// TIA Portal project "FBM_Bordeau" (V17)

(* hardware
DEVICE "S7-1200 station_1"  S7-1200 Station
   slot 0: "Rack_0"  S7-1200 Rack  Rack  V1.0
   slot 1: "PLC_1"  CPU 1214C AC/DC/Rly  6ES7 214-1BG40-0XB0  V4.5
DEVICE "S7-1200 station_2"  S7-1200 Station
   slot 0: "Rack_0"  S7-1200 Rack  Rack  V1.0
   slot 1: "PLC_2"  CPU 1214C AC/DC/Rly  6ES7 214-1BG40-0XB0  V4.5
DEVICE "HMI_1"  KTP400 Basic PN
   slot 0: "HMI_1"  KTP400 Basic PN  6AV2 123-2DB03-0AX0  17.0.0.0
   slot 1: "HMI_RT_1"  KTP400 Basic PN  6AV2 123-2DB03-0AX0  17.0.0.0
   slot 5: "HMI_1.IE_CP_1"  PROFINET Interface  17.0.0.0
      slot 1: "PROFINET Interface_1"  PROFINET Interface
         slot 1: "Port_1"  Port
*)

// ===== PLC "PLC_1"  CPU 1214C AC/DC/Rly =====

VAR_GLOBAL   // PLC tag table "Default tag table"
   "VisiteurMax" AT %MW10 : Int;
   "Alerte1" AT %MW12 : Int;
   "Alerte2" AT %MW14 : Int;
   "Occupation" AT %MW16 : Int;
   "BitAlerte1" AT %M50.0 : Bool;
   "BitAlerte2" AT %M50.1 : Bool;
   "BitNoAlerte" AT %M50.2 : Bool;
   "AnimationCarre" AT %MW18 : Int;
   "BitModifier" AT %M50.3 : Bool;
   "BitEnregistrer" AT %M50.4 : Bool;
   "BitAnnuler" AT %M50.5 : Bool;
   "AutoriseModifier" AT %M50.6 : Bool;
   "AutoriseEnregistrer" AT %M50.7 : Bool;
   "AutoriseAnnuler" AT %M51.0 : Bool;
   "FM_1" AT %M60.0 : Bool;
   "FM_2" AT %M60.1 : Bool;
   "Up" AT %M60.2 : Bool;
   "Down" AT %M60.3 : Bool;
   "FM_3" AT %M60.4 : Bool;
   "FM_4" AT %M60.5 : Bool;
   "RealOccupation" AT %MD100 : Real;
   "RealAlerte1" AT %MD104 : Real;
   "RealAlerte2" AT %MD108 : Real;
   "RealVisiteurMax" AT %MD112 : Real;
   "Tag_5" AT %MD116 : Real;
   "Tag_6" AT %MD120 : DWord;
   "FM_7" AT %M60.6 : Bool;
   "Tag_8" AT %MD122 : Real;
   "FM_9" AT %M60.7 : Bool;
   "OldVisiteurMax" AT %MW20 : Int;
   "PourcentageMax" AT %MD126 : Real;
   "PourcentageMin" AT %MD130 : Real;
   "IR1_COULOIR_1" AT %I0.0 : Bool;
   "COMPTEUR_E_COULOIR_1" AT %I0.1 : Bool;
   "COMPTEUR_S_COULOIR_1" AT %I0.2 : Bool;
   "IR1_COULOIR_2" AT %I0.3 : Bool;
   "COMPTEUR_E_COULOIR_2" AT %I0.4 : Bool;
   "COMPTEUR_S_COULOIR_2" AT %I0.5 : Bool;
   "IR1_COULOIR_3" AT %I0.6 : Bool;
   "COMPTEUR_E_COULOIR_3" AT %I0.7 : Bool;
   "COMPTEUR_S_COULOIR_3" AT %I1.0 : Bool;
   "IR1_COULOIR_4" AT %I1.1 : Bool;
   "COMPTEUR_E_COULOIR_4" AT %I1.2 : Bool;
   "COMPTEUR_S_COULOIR_4" AT %I1.3 : Bool;
   "RESERVE1" AT %I1.4 : Bool;
   "RESERVE2" AT %I1.5 : Bool;
   "COMMANDE_O_COULOIR_1" AT %Q0.0 : Bool;
   "COMMANDE_O_COULOIR_2" AT %Q0.1 : Bool;
   "COMMANDE_O_COULOIR_3" AT %Q0.2 : Bool;
   "COMMANDE_O_COULOIR_4" AT %Q0.3 : Bool;
   "COMMANDE_O_COULOIR_5" AT %Q0.4 : Bool;
   "COMMANDE_O_COULOIR_6" AT %Q0.5 : Bool;
   "COMMANDE_O_COULOIR_7" AT %Q0.6 : Bool;
   "RESERVE_SORTIE_8" AT %Q0.7 : Bool;
   "Sortie8" AT %Q1.0 : Bool;
   "Sortie9" AT %Q1.1 : Bool;
   "Clock_Byte" AT %MB0 : Byte;
   "Clock_10Hz" AT %M0.0 : Bool;
   "Clock_5Hz" AT %M0.1 : Bool;
   "Clock_2.5Hz" AT %M0.2 : Bool;
   "Clock_2Hz" AT %M0.3 : Bool;
   "Clock_1.25Hz" AT %M0.4 : Bool;
   "Clock_1Hz" AT %M0.5 : Bool;
   "Clock_0.625Hz" AT %M0.6 : Bool;
   "Clock_0.5Hz" AT %M0.7 : Bool;
   "PLC1_ImageEntree1" AT %M70.0 : Bool;
   "PLC1_ImageEntree2" AT %M70.1 : Bool;
   "PLC1_ImageEntree3" AT %M70.2 : Bool;
   "PLC1_ImageEntree4" AT %M70.3 : Bool;
   "PLC1_ImageEntree5" AT %M70.4 : Bool;
   "PLC1_ImageEntree6" AT %M70.5 : Bool;
   "PLC1_ImageEntree7" AT %M70.6 : Bool;
   "PLC1_ImageEntree8" AT %M70.7 : Bool;
   "PLC1_ImageEntree9" AT %M71.0 : Bool;
   "PLC1_ImageEntree10" AT %M71.1 : Bool;
   "PLC1_ImageEntree11" AT %M71.2 : Bool;
   "PLC1_ImageEntree12" AT %M71.3 : Bool;
   "PLC1_ImageEntree13" AT %M71.4 : Bool;
   "PLC1_ImageEntree0" AT %M71.5 : Bool;
   "SynthesEntree" AT %M71.6 : Bool;
   "SyntheseSortie" AT %M71.7 : Bool;
   "FM_SyntheseEntree" AT %M72.0 : Bool;
   "FM_SyntheseSortie" AT %M72.1 : Bool;
   "FM_IR1_C5" AT %M72.2 : Bool;
   "FM_IR1_C6" AT %M72.3 : Bool;
   "FM_IR1_C7" AT %M72.4 : Bool;
   "FM_IR1_C1" AT %M73.2 : Bool;
   "FM_IR1_C2" AT %M73.3 : Bool;
   "FM_IR1_C3" AT %M73.4 : Bool;
   "FM_IR1_C4" AT %M73.5 : Bool;
   "Tag_1" AT %M80.0 : Bool;
   "PLC1_ImageSortie0" AT %M73.6 : Bool;
   "PLC1_ImageSortie1" AT %M73.7 : Bool;
   "PLC1_ImageSortie2" AT %M74.0 : Bool;
   "PLC1_ImageSortie3" AT %M74.1 : Bool;
   "PLC1_ImageSortie4" AT %M74.2 : Bool;
   "PLC1_ImageSortie5" AT %M74.3 : Bool;
   "PLC1_ImageSortie6" AT %M74.4 : Bool;
   "PLC2_ImageSortie0" AT %M74.5 : Bool;
   "PLC2_ImageSortie1" AT %M74.6 : Bool;
   "PLC2_ImageSortie2" AT %M74.7 : Bool;
   "PLC2_ImageSortie3" AT %M75.0 : Bool;
   "PLC2_ImageSortie4" AT %M75.1 : Bool;
   "PLC2_ImageSortie5" AT %M75.2 : Bool;
   "PLC2_ImageSortie6" AT %M75.3 : Bool;
   "Tag_2" AT %M100.0 : Bool;
   "Tag_3" AT %M100.1 : Bool;
   "Tag_4" AT %M100.2 : Bool;
   "Tag_7" AT %M100.3 : Bool;
   "TEST_SORTIE" AT %M100.4 : Bool;
   "TEST_ENTREE" AT %M100.5 : Bool;
   "ResetOccupation" AT %M100.6 : Bool;
   "Tag_9" AT %M100.7 : Bool;
   "FM_COUNT_S1" AT %M103.1 : Bool;
   "Memore_Cmpt_SortieC1" AT %M101.1 : Bool;
   "TempoIR1" AT %M102.1 : Bool;
   "Tag_11" AT %I1.6 : Bool;
   "Memore_Cmpt_SortieC2" AT %M101.2 : Bool;
   "Memore_Cmpt_SortieC3" AT %M101.3 : Bool;
   "Memore_Cmpt_SortieC4" AT %M101.4 : Bool;
   "Memore_Cmpt_SortieC5" AT %M101.5 : Bool;
   "Memore_Cmpt_SortieC6" AT %M101.6 : Bool;
   "Memore_Cmpt_SortieC7" AT %M101.7 : Bool;
   "TempoIR2" AT %M102.2 : Bool;
   "TempoIR3" AT %M102.3 : Bool;
   "TempoIR4" AT %M102.4 : Bool;
   "TempoIR5" AT %M102.5 : Bool;
   "TempoIR6" AT %M102.6 : Bool;
   "TempoIR7" AT %M102.7 : Bool;
   "FM_COUNT_S2" AT %M103.2 : Bool;
   "FM_COUNT_S3" AT %M103.3 : Bool;
   "FM_COUNT_S4" AT %M103.4 : Bool;
   "FM_COUNT_S5" AT %M103.5 : Bool;
   "FM_COUNT_S6" AT %M103.6 : Bool;
   "FM_COUNT_S7" AT %M103.7 : Bool;
END_VAR

DATA_BLOCK "PLC1_DB_Bool"   // DB1
{ S7_Optimized_Access := 'FALSE' }
VERSION : 0.1
   VAR
      FM_2 : Bool;
      Up : Bool;
      FM_4 : Bool;
      FM_1 : Bool;
      AutoriseAnnuler : Bool;
      AutoriseEnregistrer : Bool;
      AutoriseModifier : Bool;
      BitAnnuler : Bool;
      Down : Bool;
      BitEnregistrer : Bool;
      BitNoAlerte : Bool;
      BitAlerte2 : Bool;
      BitAlerte1 : Bool;
      FM_7 : Bool;
      FM_9 : Bool;
      BitModifier : Bool;
      FM_3 : Bool;
   END_VAR
BEGIN
END_DATA_BLOCK

DATA_BLOCK "PLC1_DB_Real"   // DB2
{ S7_Optimized_Access := 'FALSE' }
VERSION : 0.1
   VAR
      RealOccupation : Real;
      RealAlerte1 : Real;
      RealAlerte2 : Real;
      RealVisiteurMax : Real;
      Tag_5 : Real;
      Tag_8 : Real;
      PourcentageMax : Real;
      PourcentageMin : Real;
   END_VAR
BEGIN
END_DATA_BLOCK

DATA_BLOCK "PLC1_DB_Int"   // DB3
{ S7_Optimized_Access := 'FALSE' }
VERSION : 0.1
   VAR
      OldVisiteurMax : Int;
      VisiteurMax : Int;
      AnimationCarre : Int;
      Occupation : Int;
      Alerte2 : Int;
      Alerte1 : Int;
   END_VAR
BEGIN
END_DATA_BLOCK

DATA_BLOCK "PLC1_DB_TO_GET"   // DB4
{ S7_Optimized_Access := 'FALSE' }
VERSION : 0.1
   VAR
      IR1_COULOIR_5 : Bool;
      COMPTEUR_E_COULOIR_5 : Bool;
      COMPTEUR_S_COULOIR_5 : Bool;
      IR1_COULOIR_6 : Bool;
      COMPTEUR_E_COULOIR_6 : Bool;
      COMPTEUR_S_COULOIR_6 : Bool;
      IR1_COULOIR_7 : Bool;
      COMPTEUR_E_COULOIR_7 : Bool;
      COMPTEUR_S_COULOIR_7 : Bool;
      RESERVE_ENTREE_1 : Bool;
      RESERVE_ENTREE_2 : Bool;
      RESERVE_ENTREE_3 : Bool;
      RESERVE_ENTREE_4 : Bool;
      RESERVE_ENTREE_5 : Bool;
      RESERVE_SORTIE_0 : Bool;
      RESERVE_SORTIE_1 : Bool;
      RESERVE_SORTIE_2 : Bool;
      RESERVE_SORTIE_3 : Bool;
      RESERVE_SORTIE_4 : Bool;
      RESERVE_SORTIE_5 : Bool;
      RESERVE_SORTIE_6 : Bool;
   END_VAR
BEGIN
END_DATA_BLOCK

DATA_BLOCK "PLC1_DB_TO_PUT"   // DB6
{ S7_Optimized_Access := 'FALSE' }
VERSION : 0.1
   VAR
      Entree0 : Bool;
      Entree1 : Bool;
      Entree2 : Bool;
      Entree3 : Bool;
      Entree4 : Bool;
      Entree5 : Bool;
      Entree6 : Bool;
      Entree7 : Bool;
      Entree8 : Bool;
      Entree9 : Bool;
      Entree10 : Bool;
      Entree11 : Bool;
      Entree12 : Bool;
      Entree13 : Bool;
      Sortie0 : Bool;
      Sortie1 : Bool;
      Sortie2 : Bool;
      Sortie3 : Bool;
      Sortie4 : Bool;
      Sortie5 : Bool;
      Sortie6 : Bool;
   END_VAR
BEGIN
END_DATA_BLOCK

// folder: System blocks/Program resources

DATA_BLOCK "IEC_Timer_0_DB"   // DB8
{ S7_Optimized_Access := 'TRUE' }
AUTHOR : Simatic
FAMILY : IEC
NAME : IEC_TMR
VERSION : 1.0
// stored: InstanceOfName IEC_TIMER
"IEC_TIMER"
BEGIN
END_DATA_BLOCK

DATA_BLOCK "IEC_Timer_0_DB_2"   // DB9
{ S7_Optimized_Access := 'TRUE' }
AUTHOR : Simatic
FAMILY : IEC
NAME : IEC_TMR
VERSION : 1.0
// stored: InstanceOfName IEC_TIMER
"IEC_TIMER"
BEGIN
END_DATA_BLOCK

DATA_BLOCK "IEC_Timer_0_DB_3"   // DB10
{ S7_Optimized_Access := 'TRUE' }
AUTHOR : Simatic
FAMILY : IEC
NAME : IEC_TMR
VERSION : 1.0
// stored: InstanceOfName IEC_TIMER
"IEC_TIMER"
BEGIN
END_DATA_BLOCK

DATA_BLOCK "IEC_Timer_0_DB_4"   // DB11
{ S7_Optimized_Access := 'TRUE' }
AUTHOR : Simatic
FAMILY : IEC
NAME : IEC_TMR
VERSION : 1.0
// stored: InstanceOfName IEC_TIMER
"IEC_TIMER"
BEGIN
END_DATA_BLOCK

DATA_BLOCK "IEC_Timer_0_DB_5"   // DB12
{ S7_Optimized_Access := 'TRUE' }
AUTHOR : Simatic
FAMILY : IEC
NAME : IEC_TMR
VERSION : 1.0
// stored: InstanceOfName IEC_TIMER
"IEC_TIMER"
BEGIN
END_DATA_BLOCK

DATA_BLOCK "IEC_Timer_0_DB_6"   // DB13
{ S7_Optimized_Access := 'TRUE' }
AUTHOR : Simatic
FAMILY : IEC
NAME : IEC_TMR
VERSION : 1.0
// stored: InstanceOfName IEC_TIMER
"IEC_TIMER"
BEGIN
END_DATA_BLOCK

DATA_BLOCK "IEC_Timer_0_DB_7"   // DB14
{ S7_Optimized_Access := 'TRUE' }
AUTHOR : Simatic
FAMILY : IEC
NAME : IEC_TMR
VERSION : 1.0
// stored: InstanceOfName IEC_TIMER
"IEC_TIMER"
BEGIN
END_DATA_BLOCK

DATA_BLOCK "IEC_Timer_0_DB_8"   // DB15
{ S7_Optimized_Access := 'TRUE' }
AUTHOR : Simatic
FAMILY : IEC
NAME : IEC_TMR
VERSION : 1.0
// stored: InstanceOfName IEC_TIMER
"IEC_TIMER"
BEGIN
END_DATA_BLOCK

DATA_BLOCK "IEC_Timer_0_DB_1"   // DB16
{ S7_Optimized_Access := 'TRUE' }
AUTHOR : Simatic
FAMILY : IEC
NAME : IEC_TMR
VERSION : 1.0
// stored: InstanceOfName IEC_TIMER
"IEC_TIMER"
BEGIN
END_DATA_BLOCK

DATA_BLOCK "IEC_Timer_0_DB_9"   // DB17
{ S7_Optimized_Access := 'TRUE' }
AUTHOR : Simatic
FAMILY : IEC
NAME : IEC_TMR
VERSION : 1.0
// stored: InstanceOfName IEC_TIMER
"IEC_TIMER"
BEGIN
END_DATA_BLOCK

DATA_BLOCK "IEC_Timer_0_DB_10"   // DB18
{ S7_Optimized_Access := 'TRUE' }
AUTHOR : Simatic
FAMILY : IEC
NAME : IEC_TMR
VERSION : 1.0
// stored: InstanceOfName IEC_TIMER
"IEC_TIMER"
BEGIN
END_DATA_BLOCK

DATA_BLOCK "IEC_Timer_0_DB_11"   // DB19
{ S7_Optimized_Access := 'TRUE' }
AUTHOR : Simatic
FAMILY : IEC
NAME : IEC_TMR
VERSION : 1.0
// stored: InstanceOfName IEC_TIMER
"IEC_TIMER"
BEGIN
END_DATA_BLOCK

DATA_BLOCK "IEC_Timer_0_DB_12"   // DB20
{ S7_Optimized_Access := 'TRUE' }
AUTHOR : Simatic
FAMILY : IEC
NAME : IEC_TMR
VERSION : 1.0
// stored: InstanceOfName IEC_TIMER
"IEC_TIMER"
BEGIN
END_DATA_BLOCK

DATA_BLOCK "IEC_Timer_0_DB_13"   // DB21
{ S7_Optimized_Access := 'TRUE' }
AUTHOR : Simatic
FAMILY : IEC
NAME : IEC_TMR
VERSION : 1.0
// stored: InstanceOfName IEC_TIMER
"IEC_TIMER"
BEGIN
END_DATA_BLOCK

DATA_BLOCK "IEC_Timer_0_DB_14"   // DB22
{ S7_Optimized_Access := 'TRUE' }
AUTHOR : Simatic
FAMILY : IEC
NAME : IEC_TMR
VERSION : 1.0
// stored: InstanceOfName IEC_TIMER
"IEC_TIMER"
BEGIN
END_DATA_BLOCK

DATA_BLOCK "IEC_Timer_0_DB_15"   // DB23
{ S7_Optimized_Access := 'TRUE' }
AUTHOR : Simatic
FAMILY : IEC
NAME : IEC_TMR
VERSION : 1.0
// stored: InstanceOfName IEC_TIMER
"IEC_TIMER"
BEGIN
END_DATA_BLOCK

DATA_BLOCK "IEC_Timer_0_DB_16"   // DB24
{ S7_Optimized_Access := 'TRUE' }
AUTHOR : Simatic
FAMILY : IEC
NAME : IEC_TMR
VERSION : 1.0
// stored: InstanceOfName IEC_TIMER
"IEC_TIMER"
BEGIN
END_DATA_BLOCK

DATA_BLOCK "IEC_Timer_0_DB_17"   // DB25
{ S7_Optimized_Access := 'TRUE' }
AUTHOR : Simatic
FAMILY : IEC
NAME : IEC_TMR
VERSION : 1.0
// stored: InstanceOfName IEC_TIMER
"IEC_TIMER"
BEGIN
END_DATA_BLOCK

DATA_BLOCK "IEC_Timer_0_DB_18"   // DB26
{ S7_Optimized_Access := 'TRUE' }
AUTHOR : Simatic
FAMILY : IEC
NAME : IEC_TMR
VERSION : 1.0
// stored: InstanceOfName IEC_TIMER
"IEC_TIMER"
BEGIN
END_DATA_BLOCK

DATA_BLOCK "IEC_Timer_0_DB_19"   // DB27
{ S7_Optimized_Access := 'TRUE' }
AUTHOR : Simatic
FAMILY : IEC
NAME : IEC_TMR
VERSION : 1.0
// stored: InstanceOfName IEC_TIMER
"IEC_TIMER"
BEGIN
END_DATA_BLOCK

// folder: (top level)

FUNCTION "PLC1_Get_Put_Value_PLC2" : Void   // FC1, LAD
{ S7_Optimized_Access := 'TRUE' }
VERSION : 0.1
BEGIN

REGION Network 1
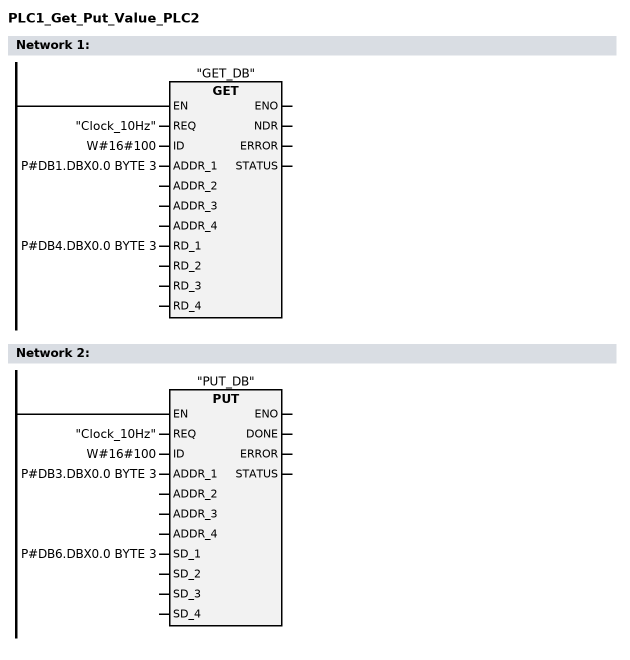
   "GET_DB"(REQ := "Clock_10Hz", ID := W#16#100, ADDR_1 := P#DB1.DBX0.0 BYTE 3, RD_1 := P#DB4.DBX0.0 BYTE 3);   // GET
END_REGION

REGION Network 2
   "PUT_DB"(REQ := "Clock_10Hz", ID := W#16#100, ADDR_1 := P#DB3.DBX0.0 BYTE 3, SD_1 := P#DB6.DBX0.0 BYTE 3);   // PUT
END_REGION
END_FUNCTION

FUNCTION "PLC1_ImageEntree" : Void   // FC2, LAD
{ S7_Optimized_Access := 'TRUE' }
VERSION : 0.1
BEGIN

REGION Network 1: SYNTHESE ENTREE SUR SITE
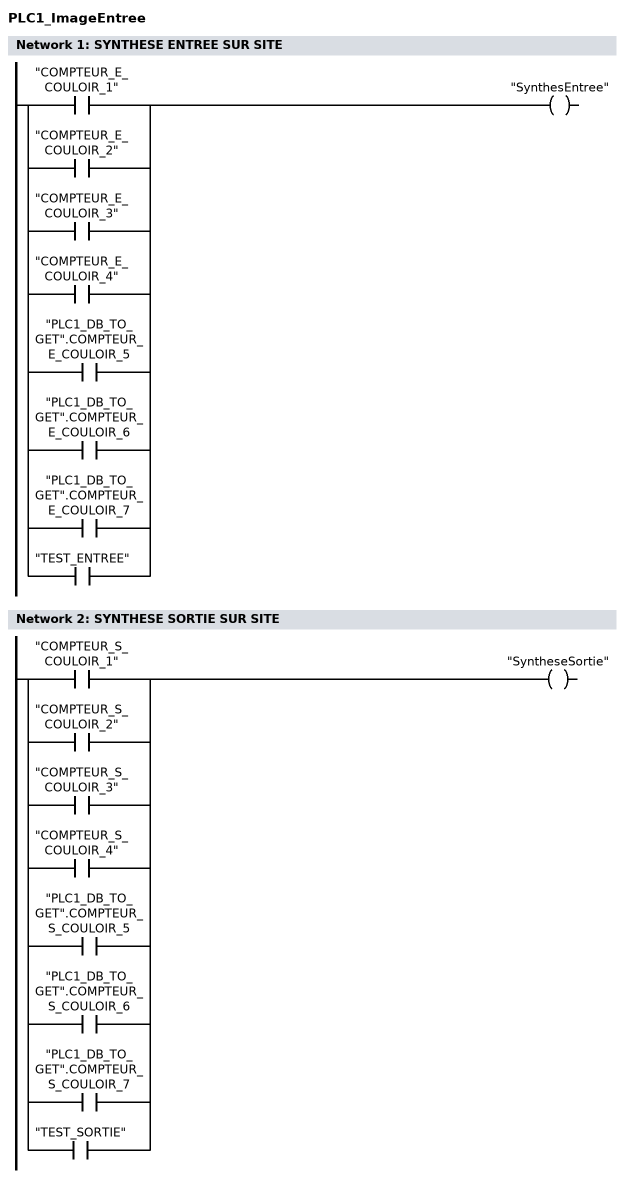
   RUNG wire#powerrail
      Contact( "COMPTEUR_E_COULOIR_1" )
      wire#w1
      Coil( "SynthesEntree" )
   END_RUNG
   RUNG wire#powerrail
      Contact( "COMPTEUR_E_COULOIR_2" )
   END_RUNG wire#w1
   RUNG wire#powerrail
      Contact( "COMPTEUR_E_COULOIR_3" )
   END_RUNG wire#w1
   RUNG wire#powerrail
      Contact( "COMPTEUR_E_COULOIR_4" )
   END_RUNG wire#w1
   RUNG wire#powerrail
      Contact( "PLC1_DB_TO_GET".COMPTEUR_E_COULOIR_5 )
   END_RUNG wire#w1
   RUNG wire#powerrail
      Contact( "PLC1_DB_TO_GET".COMPTEUR_E_COULOIR_6 )
   END_RUNG wire#w1
   RUNG wire#powerrail
      Contact( "PLC1_DB_TO_GET".COMPTEUR_E_COULOIR_7 )
   END_RUNG wire#w1
   RUNG wire#powerrail
      Contact( "TEST_ENTREE" )
   END_RUNG wire#w1
   // the same network as SCL:
   "SynthesEntree" := "COMPTEUR_E_COULOIR_1" OR "COMPTEUR_E_COULOIR_2" OR "COMPTEUR_E_COULOIR_3" OR "COMPTEUR_E_COULOIR_4" OR "PLC1_DB_TO_GET".COMPTEUR_E_COULOIR_5 OR "PLC1_DB_TO_GET".COMPTEUR_E_COULOIR_6 OR "PLC1_DB_TO_GET".COMPTEUR_E_COULOIR_7 OR "TEST_ENTREE";
END_REGION

REGION Network 2: SYNTHESE SORTIE SUR SITE
   RUNG wire#powerrail
      Contact( "COMPTEUR_S_COULOIR_1" )
      wire#w1
      Coil( "SyntheseSortie" )
   END_RUNG
   RUNG wire#powerrail
      Contact( "COMPTEUR_S_COULOIR_2" )
   END_RUNG wire#w1
   RUNG wire#powerrail
      Contact( "COMPTEUR_S_COULOIR_3" )
   END_RUNG wire#w1
   RUNG wire#powerrail
      Contact( "COMPTEUR_S_COULOIR_4" )
   END_RUNG wire#w1
   RUNG wire#powerrail
      Contact( "PLC1_DB_TO_GET".COMPTEUR_S_COULOIR_5 )
   END_RUNG wire#w1
   RUNG wire#powerrail
      Contact( "PLC1_DB_TO_GET".COMPTEUR_S_COULOIR_6 )
   END_RUNG wire#w1
   RUNG wire#powerrail
      Contact( "PLC1_DB_TO_GET".COMPTEUR_S_COULOIR_7 )
   END_RUNG wire#w1
   RUNG wire#powerrail
      Contact( "TEST_SORTIE" )
   END_RUNG wire#w1
   // the same network as SCL:
   "SyntheseSortie" := "COMPTEUR_S_COULOIR_1" OR "COMPTEUR_S_COULOIR_2" OR "COMPTEUR_S_COULOIR_3" OR "COMPTEUR_S_COULOIR_4" OR "PLC1_DB_TO_GET".COMPTEUR_S_COULOIR_5 OR "PLC1_DB_TO_GET".COMPTEUR_S_COULOIR_6 OR "PLC1_DB_TO_GET".COMPTEUR_S_COULOIR_7 OR "TEST_SORTIE";
END_REGION
END_FUNCTION

ORGANIZATION_BLOCK "PLC1_Main"   // OB1, LAD, ProgramCycle
TITLE = "Main Program Sweep (Cycle)"
{ S7_Optimized_Access := 'TRUE' }
VERSION : 0.1
   VAR_INPUT
      Initial_Call : Bool;   // Initial call of this OB
      Remanence : Bool;   // =True, if remanent data are available
   END_VAR
   VAR_TEMP   // added for the SCL form of the ladder/FBD networks
      _w1 : Bool;
      _w2 : Bool;
      _w3 : Bool;
      _w4 : Bool;
   END_VAR
BEGIN

REGION Network 1
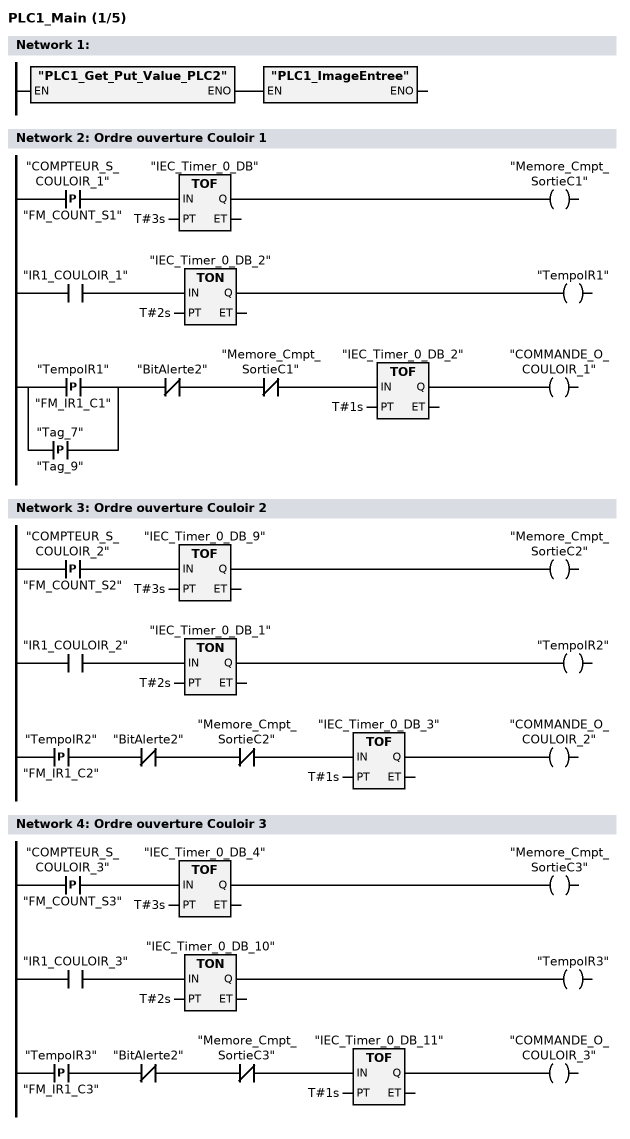
   RUNG wire#powerrail
      "PLC1_Get_Put_Value_PLC2"()
      "PLC1_ImageEntree"()
   END_RUNG
   // the same network as SCL:
   "PLC1_Get_Put_Value_PLC2"(ENO => #_w1);
   IF #_w1 THEN "PLC1_ImageEntree"(); END_IF;
END_REGION

REGION Network 2: Ordre ouverture Couloir 1
   #_w1 := "COMPTEUR_S_COULOIR_1" AND NOT "FM_COUNT_S1";   // rising edge of "COMPTEUR_S_COULOIR_1"
   "FM_COUNT_S1" := "COMPTEUR_S_COULOIR_1";
   "IEC_Timer_0_DB".TOF(IN := #_w1, PT := T#3s);
   "Memore_Cmpt_SortieC1" := "IEC_Timer_0_DB".Q;
   "IEC_Timer_0_DB_2".TON(IN := "IR1_COULOIR_1", PT := T#2s);
   "TempoIR1" := "IEC_Timer_0_DB_2".Q;
   #_w2 := "TempoIR1" AND NOT "FM_IR1_C1";   // rising edge of "TempoIR1"
   "FM_IR1_C1" := "TempoIR1";
   #_w3 := "Tag_7" AND NOT "Tag_9";   // rising edge of "Tag_7"
   "Tag_9" := "Tag_7";
   "IEC_Timer_0_DB_2".TOF(IN := (#_w2 OR #_w3) AND NOT "BitAlerte2" AND NOT "Memore_Cmpt_SortieC1", PT := T#1s);
   "COMMANDE_O_COULOIR_1" := "IEC_Timer_0_DB_2".Q;
END_REGION

REGION Network 3: Ordre ouverture Couloir 2
   #_w1 := "COMPTEUR_S_COULOIR_2" AND NOT "FM_COUNT_S2";   // rising edge of "COMPTEUR_S_COULOIR_2"
   "FM_COUNT_S2" := "COMPTEUR_S_COULOIR_2";
   "IEC_Timer_0_DB_9".TOF(IN := #_w1, PT := T#3s);
   "Memore_Cmpt_SortieC2" := "IEC_Timer_0_DB_9".Q;
   "IEC_Timer_0_DB_1".TON(IN := "IR1_COULOIR_2", PT := T#2s);
   "TempoIR2" := "IEC_Timer_0_DB_1".Q;
   #_w2 := "TempoIR2" AND NOT "FM_IR1_C2";   // rising edge of "TempoIR2"
   "FM_IR1_C2" := "TempoIR2";
   "IEC_Timer_0_DB_3".TOF(IN := #_w2 AND NOT "BitAlerte2" AND NOT "Memore_Cmpt_SortieC2", PT := T#1s);
   "COMMANDE_O_COULOIR_2" := "IEC_Timer_0_DB_3".Q;
END_REGION

REGION Network 4: Ordre ouverture Couloir 3
   #_w1 := "COMPTEUR_S_COULOIR_3" AND NOT "FM_COUNT_S3";   // rising edge of "COMPTEUR_S_COULOIR_3"
   "FM_COUNT_S3" := "COMPTEUR_S_COULOIR_3";
   "IEC_Timer_0_DB_4".TOF(IN := #_w1, PT := T#3s);
   "Memore_Cmpt_SortieC3" := "IEC_Timer_0_DB_4".Q;
   "IEC_Timer_0_DB_10".TON(IN := "IR1_COULOIR_3", PT := T#2s);
   "TempoIR3" := "IEC_Timer_0_DB_10".Q;
   #_w2 := "TempoIR3" AND NOT "FM_IR1_C3";   // rising edge of "TempoIR3"
   "FM_IR1_C3" := "TempoIR3";
   "IEC_Timer_0_DB_11".TOF(IN := #_w2 AND NOT "BitAlerte2" AND NOT "Memore_Cmpt_SortieC3", PT := T#1s);
   "COMMANDE_O_COULOIR_3" := "IEC_Timer_0_DB_11".Q;
END_REGION

REGION Network 5: Ordre ouverture Couloir 4
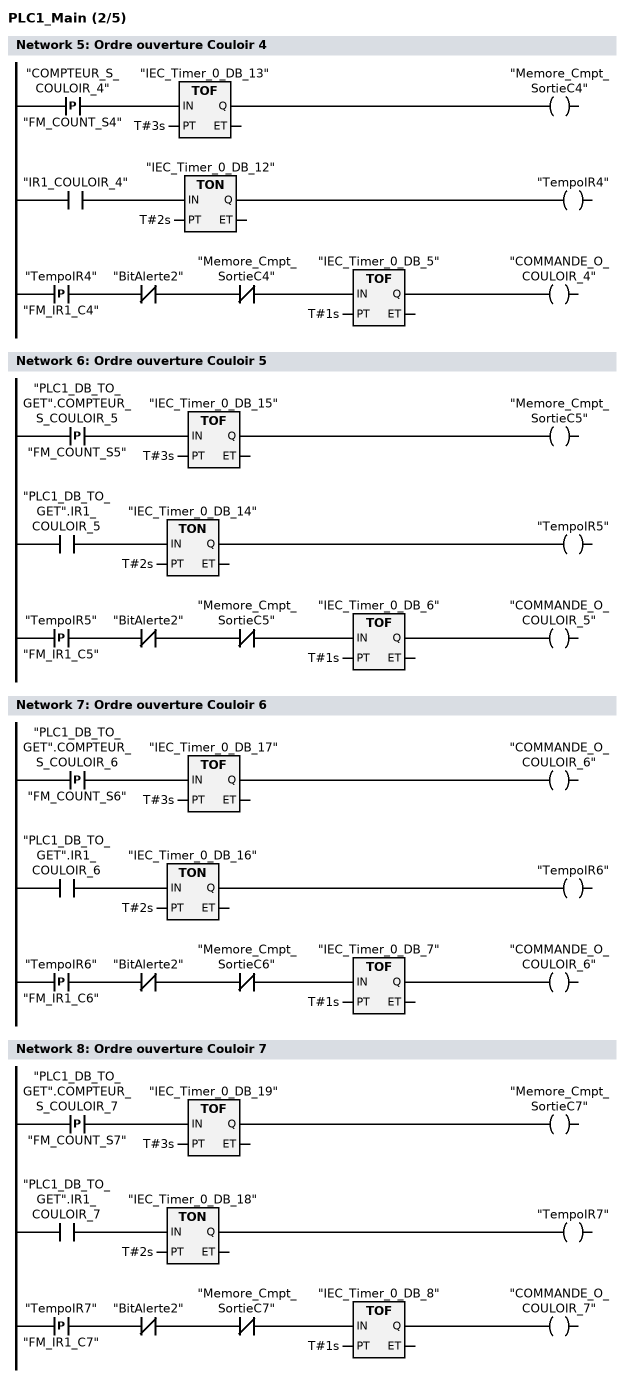
   #_w1 := "COMPTEUR_S_COULOIR_4" AND NOT "FM_COUNT_S4";   // rising edge of "COMPTEUR_S_COULOIR_4"
   "FM_COUNT_S4" := "COMPTEUR_S_COULOIR_4";
   "IEC_Timer_0_DB_13".TOF(IN := #_w1, PT := T#3s);
   "Memore_Cmpt_SortieC4" := "IEC_Timer_0_DB_13".Q;
   "IEC_Timer_0_DB_12".TON(IN := "IR1_COULOIR_4", PT := T#2s);
   "TempoIR4" := "IEC_Timer_0_DB_12".Q;
   #_w2 := "TempoIR4" AND NOT "FM_IR1_C4";   // rising edge of "TempoIR4"
   "FM_IR1_C4" := "TempoIR4";
   "IEC_Timer_0_DB_5".TOF(IN := #_w2 AND NOT "BitAlerte2" AND NOT "Memore_Cmpt_SortieC4", PT := T#1s);
   "COMMANDE_O_COULOIR_4" := "IEC_Timer_0_DB_5".Q;
END_REGION

REGION Network 6: Ordre ouverture Couloir 5
   #_w1 := "PLC1_DB_TO_GET".COMPTEUR_S_COULOIR_5 AND NOT "FM_COUNT_S5";   // rising edge of "PLC1_DB_TO_GET".COMPTEUR_S_COULOIR_5
   "FM_COUNT_S5" := "PLC1_DB_TO_GET".COMPTEUR_S_COULOIR_5;
   "IEC_Timer_0_DB_15".TOF(IN := #_w1, PT := T#3s);
   "Memore_Cmpt_SortieC5" := "IEC_Timer_0_DB_15".Q;
   "IEC_Timer_0_DB_14".TON(IN := "PLC1_DB_TO_GET".IR1_COULOIR_5, PT := T#2s);
   "TempoIR5" := "IEC_Timer_0_DB_14".Q;
   #_w2 := "TempoIR5" AND NOT "FM_IR1_C5";   // rising edge of "TempoIR5"
   "FM_IR1_C5" := "TempoIR5";
   "IEC_Timer_0_DB_6".TOF(IN := #_w2 AND NOT "BitAlerte2" AND NOT "Memore_Cmpt_SortieC5", PT := T#1s);
   "COMMANDE_O_COULOIR_5" := "IEC_Timer_0_DB_6".Q;
END_REGION

REGION Network 7: Ordre ouverture Couloir 6
   #_w1 := "PLC1_DB_TO_GET".COMPTEUR_S_COULOIR_6 AND NOT "FM_COUNT_S6";   // rising edge of "PLC1_DB_TO_GET".COMPTEUR_S_COULOIR_6
   "FM_COUNT_S6" := "PLC1_DB_TO_GET".COMPTEUR_S_COULOIR_6;
   "IEC_Timer_0_DB_17".TOF(IN := #_w1, PT := T#3s);
   "COMMANDE_O_COULOIR_6" := "IEC_Timer_0_DB_17".Q;
   "IEC_Timer_0_DB_16".TON(IN := "PLC1_DB_TO_GET".IR1_COULOIR_6, PT := T#2s);
   "TempoIR6" := "IEC_Timer_0_DB_16".Q;
   #_w2 := "TempoIR6" AND NOT "FM_IR1_C6";   // rising edge of "TempoIR6"
   "FM_IR1_C6" := "TempoIR6";
   "IEC_Timer_0_DB_7".TOF(IN := #_w2 AND NOT "BitAlerte2" AND NOT "Memore_Cmpt_SortieC6", PT := T#1s);
   "COMMANDE_O_COULOIR_6" := "IEC_Timer_0_DB_7".Q;
END_REGION

REGION Network 8: Ordre ouverture Couloir 7
   #_w1 := "PLC1_DB_TO_GET".COMPTEUR_S_COULOIR_7 AND NOT "FM_COUNT_S7";   // rising edge of "PLC1_DB_TO_GET".COMPTEUR_S_COULOIR_7
   "FM_COUNT_S7" := "PLC1_DB_TO_GET".COMPTEUR_S_COULOIR_7;
   "IEC_Timer_0_DB_19".TOF(IN := #_w1, PT := T#3s);
   "Memore_Cmpt_SortieC7" := "IEC_Timer_0_DB_19".Q;
   "IEC_Timer_0_DB_18".TON(IN := "PLC1_DB_TO_GET".IR1_COULOIR_7, PT := T#2s);
   "TempoIR7" := "IEC_Timer_0_DB_18".Q;
   #_w2 := "TempoIR7" AND NOT "FM_IR1_C7";   // rising edge of "TempoIR7"
   "FM_IR1_C7" := "TempoIR7";
   "IEC_Timer_0_DB_8".TOF(IN := #_w2 AND NOT "BitAlerte2" AND NOT "Memore_Cmpt_SortieC7", PT := T#1s);
   "COMMANDE_O_COULOIR_7" := "IEC_Timer_0_DB_8".Q;
END_REGION

REGION Network 9: Active Alerte 1
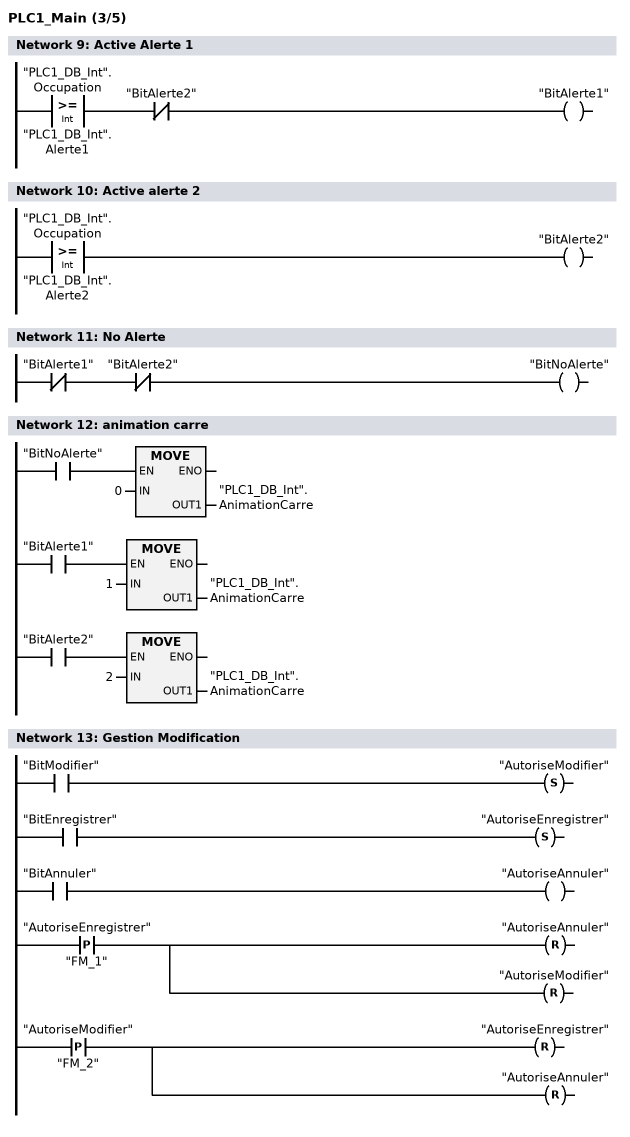
   RUNG wire#powerrail
      { S7_Templates := "SrcType := Int" } GE_Contact(in1 := "PLC1_DB_Int".Occupation, in2 := "PLC1_DB_Int".Alerte1)
      I_Contact( "BitAlerte2" )
      Coil( "BitAlerte1" )
   END_RUNG
   // the same network as SCL:
   "BitAlerte1" := ("PLC1_DB_Int".Occupation >= "PLC1_DB_Int".Alerte1) AND NOT "BitAlerte2";
END_REGION

REGION Network 10: Active alerte 2
   RUNG wire#powerrail
      { S7_Templates := "SrcType := Int" } GE_Contact(in1 := "PLC1_DB_Int".Occupation, in2 := "PLC1_DB_Int".Alerte2)
      Coil( "BitAlerte2" )
   END_RUNG
   // the same network as SCL:
   "BitAlerte2" := "PLC1_DB_Int".Occupation >= "PLC1_DB_Int".Alerte2;
END_REGION

REGION Network 11: No Alerte
   RUNG wire#powerrail
      I_Contact( "BitAlerte1" )
      I_Contact( "BitAlerte2" )
      Coil( "BitNoAlerte" )
   END_RUNG
   // the same network as SCL:
   "BitNoAlerte" := NOT "BitAlerte1" AND NOT "BitAlerte2";
END_REGION

REGION Network 12: animation carre
   RUNG wire#powerrail
      Contact( "BitNoAlerte" )
      Move(in := 0, out1 => "PLC1_DB_Int".AnimationCarre)
   END_RUNG
   RUNG wire#powerrail
      Contact( "BitAlerte1" )
      Move(in := 1, out1 => "PLC1_DB_Int".AnimationCarre)
   END_RUNG
   RUNG wire#powerrail
      Contact( "BitAlerte2" )
      Move(in := 2, out1 => "PLC1_DB_Int".AnimationCarre)
   END_RUNG
   // the same network as SCL:
   IF "BitNoAlerte" THEN "PLC1_DB_Int".AnimationCarre := 0; END_IF;
   IF "BitAlerte1" THEN "PLC1_DB_Int".AnimationCarre := 1; END_IF;
   IF "BitAlerte2" THEN "PLC1_DB_Int".AnimationCarre := 2; END_IF;
END_REGION

REGION Network 13: Gestion Modification
   RUNG wire#powerrail
      Contact( "BitModifier" )
      S_Coil( "AutoriseModifier" )
   END_RUNG
   RUNG wire#powerrail
      Contact( "BitEnregistrer" )
      S_Coil( "AutoriseEnregistrer" )
   END_RUNG
   RUNG wire#powerrail
      Contact( "BitAnnuler" )
      Coil( "AutoriseAnnuler" )
   END_RUNG
   RUNG wire#powerrail
      P_Contact(operand := "AutoriseEnregistrer", bit := "FM_1")
      wire#w1
      R_Coil( "AutoriseAnnuler" )
   END_RUNG
   RUNG wire#w1
      R_Coil( "AutoriseModifier" )
   END_RUNG
   RUNG wire#powerrail
      P_Contact(operand := "AutoriseModifier", bit := "FM_2")
      wire#w2
      R_Coil( "AutoriseEnregistrer" )
   END_RUNG
   RUNG wire#w2
      R_Coil( "AutoriseAnnuler" )
   END_RUNG
   // the same network as SCL:
   IF "BitModifier" THEN "AutoriseModifier" := TRUE; END_IF;
   IF "BitEnregistrer" THEN "AutoriseEnregistrer" := TRUE; END_IF;
   "AutoriseAnnuler" := "BitAnnuler";
   #_w1 := "AutoriseEnregistrer" AND NOT "FM_1";   // rising edge of "AutoriseEnregistrer"
   "FM_1" := "AutoriseEnregistrer";
   IF #_w1 THEN
       "AutoriseAnnuler" := FALSE;
       "AutoriseModifier" := FALSE;
   END_IF;
   #_w2 := "AutoriseModifier" AND NOT "FM_2";   // rising edge of "AutoriseModifier"
   "FM_2" := "AutoriseModifier";
   IF #_w2 THEN
       "AutoriseEnregistrer" := FALSE;
       "AutoriseAnnuler" := FALSE;
   END_IF;
END_REGION

REGION Network 14: Gestion de Loccupation du site
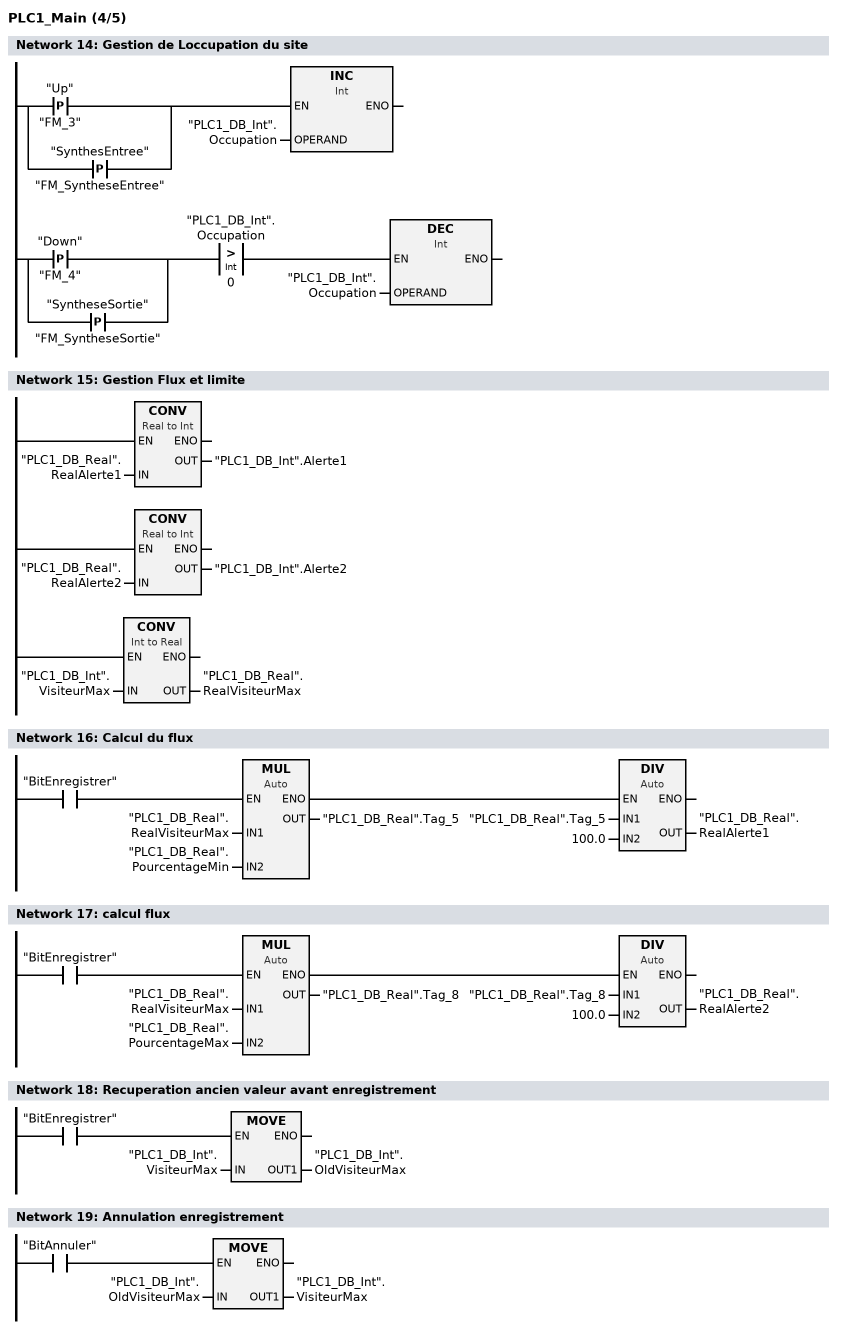
   RUNG wire#powerrail
      P_Contact(operand := "Up", bit := "FM_3")
      wire#w1
      { S7_Templates := "DestType := Int" } Inc( "PLC1_DB_Int".Occupation )
   END_RUNG
   RUNG wire#powerrail
      P_Contact(operand := "SynthesEntree", bit := "FM_SyntheseEntree")
   END_RUNG wire#w1
   RUNG wire#powerrail
      P_Contact(operand := "Down", bit := "FM_4")
      wire#w2
      { S7_Templates := "SrcType := Int" } GT_Contact(in1 := "PLC1_DB_Int".Occupation, in2 := 0)
      { S7_Templates := "DestType := Int" } Dec( "PLC1_DB_Int".Occupation )
   END_RUNG
   RUNG wire#powerrail
      P_Contact(operand := "SyntheseSortie", bit := "FM_SyntheseSortie")
   END_RUNG wire#w2
   // the same network as SCL:
   #_w1 := "Up" AND NOT "FM_3";   // rising edge of "Up"
   "FM_3" := "Up";
   #_w2 := "SynthesEntree" AND NOT "FM_SyntheseEntree";   // rising edge of "SynthesEntree"
   "FM_SyntheseEntree" := "SynthesEntree";
   IF #_w1 OR #_w2 THEN "PLC1_DB_Int".Occupation := "PLC1_DB_Int".Occupation + 1; END_IF;
   #_w3 := "Down" AND NOT "FM_4";   // rising edge of "Down"
   "FM_4" := "Down";
   #_w4 := "SyntheseSortie" AND NOT "FM_SyntheseSortie";   // rising edge of "SyntheseSortie"
   "FM_SyntheseSortie" := "SyntheseSortie";
   IF (#_w3 OR #_w4) AND ("PLC1_DB_Int".Occupation > 0) THEN
       "PLC1_DB_Int".Occupation := "PLC1_DB_Int".Occupation - 1;
   END_IF;
END_REGION

REGION Network 15: Gestion Flux et limite
   RUNG wire#powerrail
      { S7_Templates := "[SrcType := Real, DestType := Int]" } Convert(in := "PLC1_DB_Real".RealAlerte1, out => "PLC1_DB_Int".Alerte1)
   END_RUNG
   RUNG wire#powerrail
      { S7_Templates := "[SrcType := Real, DestType := Int]" } Convert(in := "PLC1_DB_Real".RealAlerte2, out => "PLC1_DB_Int".Alerte2)
   END_RUNG
   RUNG wire#powerrail
      { S7_Templates := "[SrcType := Int, DestType := Real]" } Convert(in := "PLC1_DB_Int".VisiteurMax, out => "PLC1_DB_Real".RealVisiteurMax)
   END_RUNG
   // the same network as SCL:
   "PLC1_DB_Int".Alerte1 := REAL_TO_INT("PLC1_DB_Real".RealAlerte1);
   "PLC1_DB_Int".Alerte2 := REAL_TO_INT("PLC1_DB_Real".RealAlerte2);
   "PLC1_DB_Real".RealVisiteurMax := INT_TO_REAL("PLC1_DB_Int".VisiteurMax);
END_REGION

REGION Network 16: Calcul du flux
   RUNG wire#powerrail
      Contact( "BitEnregistrer" )
      Mul(in1 := "PLC1_DB_Real".RealVisiteurMax, in2 := "PLC1_DB_Real".PourcentageMin, out => "PLC1_DB_Real".Tag_5)
      Div(in1 := "PLC1_DB_Real".Tag_5, in2 := 100.0, out => "PLC1_DB_Real".RealAlerte1)
   END_RUNG
   // the same network as SCL:
   IF "BitEnregistrer" THEN
       "PLC1_DB_Real".Tag_5 := "PLC1_DB_Real".RealVisiteurMax * "PLC1_DB_Real".PourcentageMin;
       "PLC1_DB_Real".RealAlerte1 := "PLC1_DB_Real".Tag_5 / 100.0;
   END_IF;
END_REGION

REGION Network 17: calcul flux
   RUNG wire#powerrail
      Contact( "BitEnregistrer" )
      Mul(in1 := "PLC1_DB_Real".RealVisiteurMax, in2 := "PLC1_DB_Real".PourcentageMax, out => "PLC1_DB_Real".Tag_8)
      Div(in1 := "PLC1_DB_Real".Tag_8, in2 := 100.0, out => "PLC1_DB_Real".RealAlerte2)
   END_RUNG
   // the same network as SCL:
   IF "BitEnregistrer" THEN
       "PLC1_DB_Real".Tag_8 := "PLC1_DB_Real".RealVisiteurMax * "PLC1_DB_Real".PourcentageMax;
       "PLC1_DB_Real".RealAlerte2 := "PLC1_DB_Real".Tag_8 / 100.0;
   END_IF;
END_REGION

REGION Network 18: Recuperation ancien valeur avant enregistrement
   RUNG wire#powerrail
      Contact( "BitEnregistrer" )
      Move(in := "PLC1_DB_Int".VisiteurMax, out1 => "PLC1_DB_Int".OldVisiteurMax)
   END_RUNG
   // the same network as SCL:
   IF "BitEnregistrer" THEN "PLC1_DB_Int".OldVisiteurMax := "PLC1_DB_Int".VisiteurMax; END_IF;
END_REGION

REGION Network 19: Annulation enregistrement
   RUNG wire#powerrail
      Contact( "BitAnnuler" )
      Move(in := "PLC1_DB_Int".OldVisiteurMax, out1 => "PLC1_DB_Int".VisiteurMax)
   END_RUNG
   // the same network as SCL:
   IF "BitAnnuler" THEN "PLC1_DB_Int".VisiteurMax := "PLC1_DB_Int".OldVisiteurMax; END_IF;
END_REGION

REGION Network 20
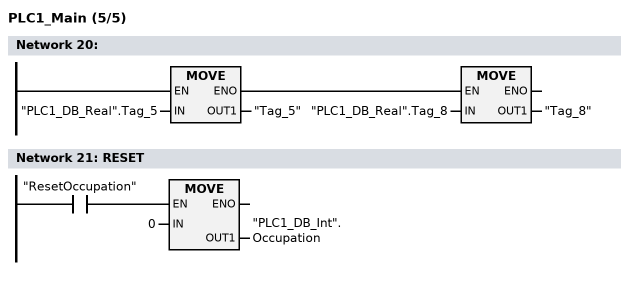
   RUNG wire#powerrail
      Move(in := "PLC1_DB_Real".Tag_5, out1 => "Tag_5")
      Move(in := "PLC1_DB_Real".Tag_8, out1 => "Tag_8")
   END_RUNG
   // the same network as SCL:
   "Tag_5" := "PLC1_DB_Real".Tag_5;
   "Tag_8" := "PLC1_DB_Real".Tag_8;
END_REGION

REGION Network 21: RESET
   RUNG wire#powerrail
      Contact( "ResetOccupation" )
      Move(in := 0, out1 => "PLC1_DB_Int".Occupation)
   END_RUNG
   // the same network as SCL:
   IF "ResetOccupation" THEN "PLC1_DB_Int".Occupation := 0; END_IF;
END_REGION
END_ORGANIZATION_BLOCK

ORGANIZATION_BLOCK "PLC1_Startup"   // OB100, LAD, Startup
TITLE = "Complete Restart"
{ S7_Optimized_Access := 'TRUE' }
VERSION : 0.1
   VAR_INPUT
      LostRetentive : Bool;   // True if retentive data are lost
      LostRTC : Bool;   // True if date and time are lost
   END_VAR
BEGIN

REGION Network 1
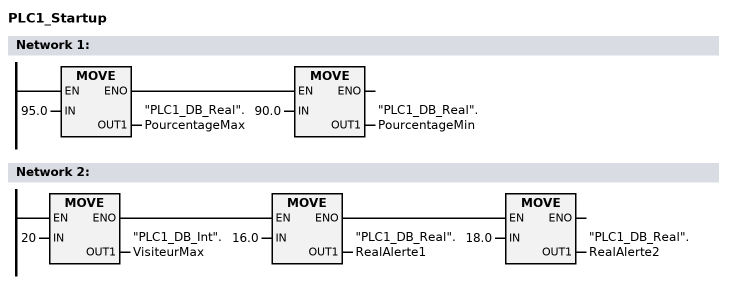
   RUNG wire#powerrail
      Move(in := 95.0, out1 => "PLC1_DB_Real".PourcentageMax)
      Move(in := 90.0, out1 => "PLC1_DB_Real".PourcentageMin)
   END_RUNG
   // the same network as SCL:
   "PLC1_DB_Real".PourcentageMax := 95.0;
   "PLC1_DB_Real".PourcentageMin := 90.0;
END_REGION

REGION Network 2
   RUNG wire#powerrail
      Move(in := 20, out1 => "PLC1_DB_Int".VisiteurMax)
      Move(in := 16.0, out1 => "PLC1_DB_Real".RealAlerte1)
      Move(in := 18.0, out1 => "PLC1_DB_Real".RealAlerte2)
   END_RUNG
   // the same network as SCL:
   "PLC1_DB_Int".VisiteurMax := 20;
   "PLC1_DB_Real".RealAlerte1 := 16.0;
   "PLC1_DB_Real".RealAlerte2 := 18.0;
END_REGION
END_ORGANIZATION_BLOCK

// ===== PLC "PLC_2"  CPU 1214C AC/DC/Rly =====

VAR_GLOBAL   // PLC tag table "Default tag table"
   "Entree0" AT %I0.0 : Bool;
   "Entree1" AT %I0.1 : Bool;
   "Entree2" AT %I0.2 : Bool;
   "Entree3" AT %I0.3 : Bool;
   "Entree4" AT %I0.4 : Bool;
   "Entree5" AT %I0.5 : Bool;
   "Entree6" AT %I0.6 : Bool;
   "Entree7" AT %I0.7 : Bool;
   "Entree8" AT %I1.0 : Bool;
   "Entree9" AT %I1.1 : Bool;
   "Entree10" AT %I1.2 : Bool;
   "Entree11" AT %I1.3 : Bool;
   "Entree12" AT %I1.4 : Bool;
   "Entree13" AT %I1.5 : Bool;
   "Sortie0" AT %Q0.0 : Bool;
   "Sortie1" AT %Q0.1 : Bool;
   "Sortie2" AT %Q0.2 : Bool;
   "Sortie3" AT %Q0.3 : Bool;
   "Sortie4" AT %Q0.4 : Bool;
   "Sortie5" AT %Q0.5 : Bool;
   "Sortie6" AT %Q0.6 : Bool;
   "Sortie7" AT %Q0.7 : Bool;
   "Sortie8" AT %Q1.0 : Bool;
   "Sortie9" AT %Q1.1 : Bool;
   "Clock_Byte" AT %MB0 : Byte;
   "Clock_10Hz" AT %M0.0 : Bool;
   "Clock_5Hz" AT %M0.1 : Bool;
   "Clock_2.5Hz" AT %M0.2 : Bool;
   "Clock_2Hz" AT %M0.3 : Bool;
   "Clock_1.25Hz" AT %M0.4 : Bool;
   "Clock_1Hz" AT %M0.5 : Bool;
   "Clock_0.625Hz" AT %M0.6 : Bool;
   "Clock_0.5Hz" AT %M0.7 : Bool;
   "Tag_1" AT %M50.0 : Bool;
   "Tag_2" AT %M80.0 : Bool;
   "Tag_3" AT %M100.1 : Bool;
   "Tag_4" AT %M100.2 : Bool;
   "Tag_5" AT %M100.3 : Bool;
END_VAR

DATA_BLOCK "PLC2_DB_TO_PUT"   // DB1
{ S7_Optimized_Access := 'FALSE' }
VERSION : 0.1
   VAR
      Entree0 : Bool;
      Entree1 : Bool;
      Entree2 : Bool;
      Entree3 : Bool;
      Entree4 : Bool;
      Entree5 : Bool;
      Entree6 : Bool;
      Entree7 : Bool;
      Entree8 : Bool;
      Entree9 : Bool;
      Entree10 : Bool;
      Entree11 : Bool;
      Entree12 : Bool;
      Entree13 : Bool;
      Sortie0 : Bool;
      Sortie1 : Bool;
      Sortie2 : Bool;
      Sortie3 : Bool;
      Sortie4 : Bool;
      Sortie5 : Bool;
      Sortie6 : Bool;
   END_VAR
BEGIN
END_DATA_BLOCK

DATA_BLOCK "PLC2_DB_TO_GET"   // DB3
{ S7_Optimized_Access := 'FALSE' }
VERSION : 0.1
   VAR
      Entree0 : Bool;
      Entree1 : Bool;
      Entree2 : Bool;
      Entree3 : Bool;
      Entree4 : Bool;
      Entree5 : Bool;
      Entree6 : Bool;
      Entree7 : Bool;
      Entree8 : Bool;
      Entree9 : Bool;
      Entree10 : Bool;
      Entree11 : Bool;
      Entree12 : Bool;
      Entree13 : Bool;
      Sortie0 : Bool;
      Sortie1 : Bool;
      Sortie2 : Bool;
      Sortie3 : Bool;
      Sortie4 : Bool;
      Sortie5 : Bool;
      Sortie6 : Bool;
   END_VAR
BEGIN
END_DATA_BLOCK

FUNCTION "PLC2_Put_Get_Value_PLC1" : Void   // FC1, LAD
{ S7_Optimized_Access := 'TRUE' }
VERSION : 0.1
BEGIN

REGION Network 1
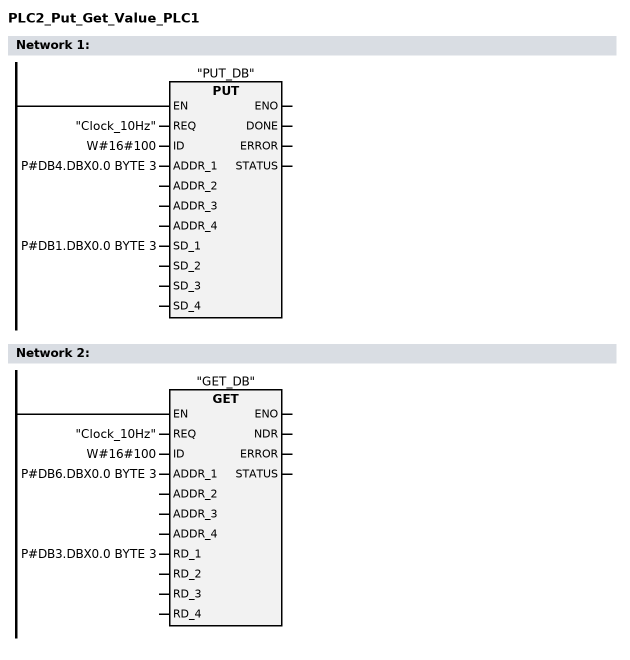
   "PUT_DB"(REQ := "Clock_10Hz", ID := W#16#100, ADDR_1 := P#DB4.DBX0.0 BYTE 3, SD_1 := P#DB1.DBX0.0 BYTE 3);   // PUT
END_REGION

REGION Network 2
   "GET_DB"(REQ := "Clock_10Hz", ID := W#16#100, ADDR_1 := P#DB6.DBX0.0 BYTE 3, RD_1 := P#DB3.DBX0.0 BYTE 3);   // GET
END_REGION
END_FUNCTION

ORGANIZATION_BLOCK "PLC2_Main"   // OB1, LAD, ProgramCycle
TITLE = "Main Program Sweep (Cycle)"
{ S7_Optimized_Access := 'TRUE' }
VERSION : 0.1
   VAR_INPUT
      Initial_Call : Bool;   // Initial call of this OB
      Remanence : Bool;   // =True, if remanent data are available
   END_VAR
BEGIN

REGION Network 1
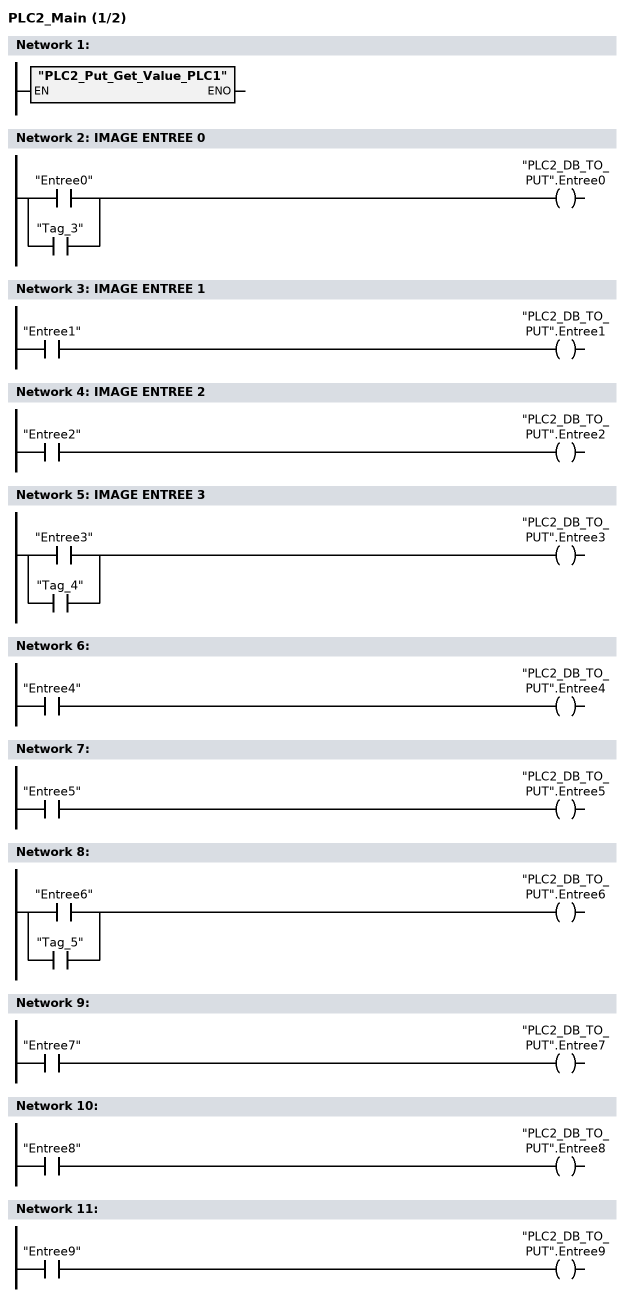
   RUNG wire#powerrail
      "PLC2_Put_Get_Value_PLC1"()
   END_RUNG
   // the same network as SCL:
   "PLC2_Put_Get_Value_PLC1"();
END_REGION

REGION Network 2: IMAGE ENTREE 0
   RUNG wire#powerrail
      Contact( "Entree0" )
      wire#w1
      Coil( "PLC2_DB_TO_PUT".Entree0 )
   END_RUNG
   RUNG wire#powerrail
      Contact( "Tag_3" )
   END_RUNG wire#w1
   // the same network as SCL:
   "PLC2_DB_TO_PUT".Entree0 := "Entree0" OR "Tag_3";
END_REGION

REGION Network 3: IMAGE ENTREE 1
   RUNG wire#powerrail
      Contact( "Entree1" )
      Coil( "PLC2_DB_TO_PUT".Entree1 )
   END_RUNG
   // the same network as SCL:
   "PLC2_DB_TO_PUT".Entree1 := "Entree1";
END_REGION

REGION Network 4: IMAGE ENTREE 2
   RUNG wire#powerrail
      Contact( "Entree2" )
      Coil( "PLC2_DB_TO_PUT".Entree2 )
   END_RUNG
   // the same network as SCL:
   "PLC2_DB_TO_PUT".Entree2 := "Entree2";
END_REGION

REGION Network 5: IMAGE ENTREE 3
   RUNG wire#powerrail
      Contact( "Entree3" )
      wire#w1
      Coil( "PLC2_DB_TO_PUT".Entree3 )
   END_RUNG
   RUNG wire#powerrail
      Contact( "Tag_4" )
   END_RUNG wire#w1
   // the same network as SCL:
   "PLC2_DB_TO_PUT".Entree3 := "Entree3" OR "Tag_4";
END_REGION

REGION Network 6
   RUNG wire#powerrail
      Contact( "Entree4" )
      Coil( "PLC2_DB_TO_PUT".Entree4 )
   END_RUNG
   // the same network as SCL:
   "PLC2_DB_TO_PUT".Entree4 := "Entree4";
END_REGION

REGION Network 7
   RUNG wire#powerrail
      Contact( "Entree5" )
      Coil( "PLC2_DB_TO_PUT".Entree5 )
   END_RUNG
   // the same network as SCL:
   "PLC2_DB_TO_PUT".Entree5 := "Entree5";
END_REGION

REGION Network 8
   RUNG wire#powerrail
      Contact( "Entree6" )
      wire#w1
      Coil( "PLC2_DB_TO_PUT".Entree6 )
   END_RUNG
   RUNG wire#powerrail
      Contact( "Tag_5" )
   END_RUNG wire#w1
   // the same network as SCL:
   "PLC2_DB_TO_PUT".Entree6 := "Entree6" OR "Tag_5";
END_REGION

REGION Network 9
   RUNG wire#powerrail
      Contact( "Entree7" )
      Coil( "PLC2_DB_TO_PUT".Entree7 )
   END_RUNG
   // the same network as SCL:
   "PLC2_DB_TO_PUT".Entree7 := "Entree7";
END_REGION

REGION Network 10
   RUNG wire#powerrail
      Contact( "Entree8" )
      Coil( "PLC2_DB_TO_PUT".Entree8 )
   END_RUNG
   // the same network as SCL:
   "PLC2_DB_TO_PUT".Entree8 := "Entree8";
END_REGION

REGION Network 11
   RUNG wire#powerrail
      Contact( "Entree9" )
      Coil( "PLC2_DB_TO_PUT".Entree9 )
   END_RUNG
   // the same network as SCL:
   "PLC2_DB_TO_PUT".Entree9 := "Entree9";
END_REGION

REGION Network 12
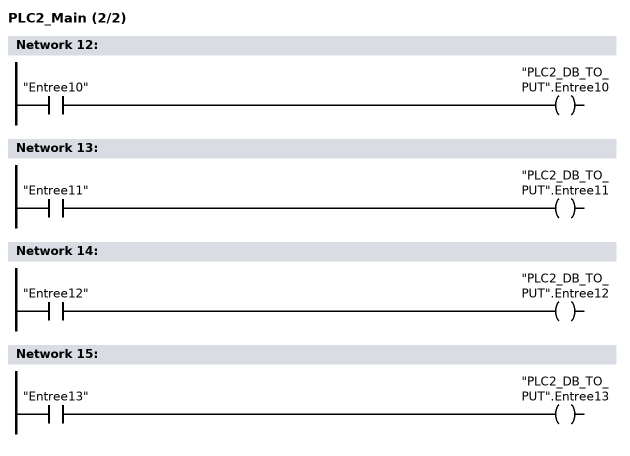
   RUNG wire#powerrail
      Contact( "Entree10" )
      Coil( "PLC2_DB_TO_PUT".Entree10 )
   END_RUNG
   // the same network as SCL:
   "PLC2_DB_TO_PUT".Entree10 := "Entree10";
END_REGION

REGION Network 13
   RUNG wire#powerrail
      Contact( "Entree11" )
      Coil( "PLC2_DB_TO_PUT".Entree11 )
   END_RUNG
   // the same network as SCL:
   "PLC2_DB_TO_PUT".Entree11 := "Entree11";
END_REGION

REGION Network 14
   RUNG wire#powerrail
      Contact( "Entree12" )
      Coil( "PLC2_DB_TO_PUT".Entree12 )
   END_RUNG
   // the same network as SCL:
   "PLC2_DB_TO_PUT".Entree12 := "Entree12";
END_REGION

REGION Network 15
   RUNG wire#powerrail
      Contact( "Entree13" )
      Coil( "PLC2_DB_TO_PUT".Entree13 )
   END_RUNG
   // the same network as SCL:
   "PLC2_DB_TO_PUT".Entree13 := "Entree13";
END_REGION
END_ORGANIZATION_BLOCK

(* ===== HMI "HMI_RT_1" =====
system functions are stored by id; their names below are inferred from use
connection "HMI_Connection_1": ETHERNET, SMART_S7_1200_OMS

HMI tags "Default tag table"
   "VisiteurMax" : Int = PLC VisiteurMax AT %MW10, 1 s
   "Alerte1" : Int = PLC Alerte1 AT %MW12, 1 s
   "Alerte2" : Int = PLC Alerte2 AT %MW14, 1 s
   "Occupation" : Int = PLC Occupation AT %MW16, 1 s
   "BitAlerte1" : Bool = PLC BitAlerte1 AT %M50.0, 1 s
   "BitAlerte2" : Bool = PLC BitAlerte2 AT %M50.1, 1 s
   "BitNoAlerte" : Bool = PLC BitNoAlerte AT %M50.2, 1 s
   "AnimationCarre" : Int = PLC AnimationCarre AT %MW18, 1 s
   "BitModifier" : Bool = PLC BitModifier AT %M50.3, 1 s
   "BitEnregistrer" : Bool = PLC BitEnregistrer AT %M50.4, 1 s
   "BitAnnuler" : Bool = PLC BitAnnuler AT %M50.5, 1 s
   "AutoriseEnregistrer" : Bool = PLC AutoriseEnregistrer AT %M50.7, 1 s
   "AutoriseAnnuler" : Bool = PLC AutoriseAnnuler AT %M51.0, 1 s
   "AutoriseModifier" : Bool = PLC AutoriseModifier AT %M50.6, 1 s
   "Up" : Bool = PLC Up AT %M60.2, 1 s
   "Down" : Bool = PLC Down AT %M60.3, 1 s
   "PourcentageMax" : Real = PLC PourcentageMax AT %MD126, 1 s
   "PourcentageMin" : Real = PLC PourcentageMin AT %MD130, 1 s
   "DB_Real_RealOccupation" : Real = PLC PLC1_DB_Real.RealOccupation AT %DB2.DBD0, 1 s
   "DB_Real_RealAlerte1" : Real = PLC PLC1_DB_Real.RealAlerte1 AT %DB2.DBD4, 1 s
   "DB_Real_RealAlerte2" : Real = PLC PLC1_DB_Real.RealAlerte2 AT %DB2.DBD8, 1 s
   "DB_Real_RealVisiteurMax" : Real = PLC PLC1_DB_Real.RealVisiteurMax AT %DB2.DBD12, 1 s
   "DB_Real_Tag_5" : Real = PLC PLC1_DB_Real.Tag_5 AT %DB2.DBD16, 1 s
   "DB_Real_Tag_8" : Real = PLC PLC1_DB_Real.Tag_8 AT %DB2.DBD20, 1 s
   "DB_Real_PourcentageMax" : Real = PLC PLC1_DB_Real.PourcentageMax AT %DB2.DBD24, 1 s
   "DB_Real_PourcentageMin" : Real = PLC PLC1_DB_Real.PourcentageMin AT %DB2.DBD28, 1 s
   "DB_Int_OldVisiteurMax" : Int = PLC PLC1_DB_Int.OldVisiteurMax AT %DB3.DBW0, 1 s
   "DB_Int_VisiteurMax" : Int = PLC PLC1_DB_Int.VisiteurMax AT %DB3.DBW2, 1 s
   "DB_Int_AnimationCarre" : Int = PLC PLC1_DB_Int.AnimationCarre AT %DB3.DBW4, 1 s
   "DB_Int_Occupation" : Int = PLC PLC1_DB_Int.Occupation AT %DB3.DBW6, 1 s
   "DB_Int_Alerte2" : Int = PLC PLC1_DB_Int.Alerte2 AT %DB3.DBW8, 1 s
   "DB_Int_Alerte1" : Int = PLC PLC1_DB_Int.Alerte1 AT %DB3.DBW10, 1 s
   "ResetOccupation" : Bool = PLC ResetOccupation AT %M100.6, 1 s

Template "Template_1" 480x272
   Button "Exit" at 714,429 size 71x50; TextOff 'Exit'; PictureOff "ExitRuntime_KTP700_Basic_PN_TR"; PictureOn "ExitRuntime_KTP700_Basic_PN_TR"
      on Release: StopRuntime(0)
   Button "Template_Button" at 614,429 size 71x50; TextOff 'Text'
   Button "Template_Button_1" at 514,429 size 71x50; TextOff 'Text'
   Button "Template_Button_2" at 414,429 size 71x50; TextOff 'Text'
   Button "Template_Button_3" at 314,429 size 71x50; TextOff 'Text'
   Button "Template_Button_4" at 214,429 size 71x50; TextOff 'Text'
   Button "Template_Button_5" at 114,429 size 71x50; TextOff 'Text'
   Button "Start screen" at 14,429 size 71x50; TextOff 'Start screen'; PictureOff "NavigateHome_KTP700_Basic_PN_TR"; PictureOn "NavigateHome_KTP700_Basic_PN_TR"
      on Release: ActivateScreen("Main", 0)

screen "Main" 480x272, template "Template_1"
   Rectangle "Rectangle_6" at 234,155 size 138x58
      Visibility <- "AutoriseModifier"
   Rectangle "Rectangle_7" at 219,216 size 166x89
      Visibility <- "AutoriseModifier"
   Rectangle "Rectangle_5" at 337,58 size 138x149
      Appearance <- "DB_Int_AnimationCarre"
   Group "Group_1" at 345,211 size 56x57; Picture "Up_Arrow"
   Group "Group_2" at 414,211 size 55x58; Picture "Down_Arrow"
   GraphicView "Graphic view_6" at 301,0 size 178x35; Picture "LogoFBMACASYSTEM"
   GraphicView "Graphic view_3" at 356,99 size 99x71; Picture "AlerteImage"
      Visibility <- "BitAlerte2"
   GraphicView "Graphic view_1" at 356,99 size 99x71; Picture "WarningImage"
      Visibility <- "BitAlerte1"
   GraphicView "Graphic view_2" at 356,99 size 99x71; Picture "CheckImage"
      Visibility <- "BitNoAlerte"
   TextField "Text field_1" at 8,108 size 148x29; Text 'Visiteurs max'
   TextField "Text field_2" at 11,29 size 136x32; Text 'Occupation'
   TextField "Text field_3" at 13,158 size 86x29; Text 'Alerte 1'
   TextField "Text field_4" at 16,191 size 86x29; Text 'Alerte 2'
   IOField "I/O field_2" at 150,20 size 114x48; FormatPattern 99999
      ProcessValue <- "DB_Int_Occupation"
   Button "Button_1" at 104,240 size 70x26; TextOff 'Modifier'; Authorization "User administration"
      on Press: function_b14e0dd5("BitModifier", 0)
      Appearance <- "AutoriseModifier"
   Button "Button_2" at 186,239 size 82x27; TextOff 'Enregistrer'
      on Press: function_b14e0dd5("BitEnregistrer", 0); function_f23ef4c9()
      Visibility <- "AutoriseModifier"
   Button "Button_3" at 18,239 size 68x27; TextOff 'Annuler'
      on Press: function_b14e0dd5("BitAnnuler", 0); function_f23ef4c9()
      Visibility <- "AutoriseModifier"
   IOField "I/O field_1" at 169,103 size 86x37; FormatPattern 99999
      ProcessValue <- "DB_Int_VisiteurMax"
   IOField "I/O field_3" at 176,153 size 81x32; FormatPattern 99999
      ProcessValue <- "DB_Int_Alerte1"
   IOField "I/O field_4" at 177,192 size 81x32; FormatPattern 99999
      ProcessValue <- "DB_Int_Alerte2"
   IOField "I/O field_5" at 289,201 size 46x32; FormatPattern 99
      Visibility <- "AutoriseModifier"
      ProcessValue <- "DB_Real_PourcentageMax"
   IOField "I/O field_6" at 288,163 size 49x32; FormatPattern 99
      Visibility <- "AutoriseModifier"
      ProcessValue <- "DB_Real_PourcentageMin"
   Rectangle "Rectangle_1" at 162,97 size 101x50
      Visibility <- "AutoriseModifier"
   Button "Button_6" at 343,219 size 126x40; TextOff 'RESET'
      Visibility <- "AutoriseModifier"
      on Press: function_b14e0dd5("ResetOccupation", 0)
   Button "Button_4" at 345,211 size 56x57; TextOff 'Text'
      on Press: function_b14e0dd5("Up", 0)
      Visibility <- "AutoriseModifier"
   GraphicView "Graphic view_4" at 358,240 size 30x25; Picture "Up_Arrow"
      Visibility <- "AutoriseModifier"
   Button "Button_5" at 414,211 size 55x58; TextOff 'Text'
      on Press: function_b14e0dd5("Down", 0)
      Visibility <- "AutoriseModifier"
   GraphicView "Graphic view_5" at 427,240 size 30x26; Picture "Down_Arrow"
      Visibility <- "AutoriseModifier"

screen "Screen_1" 480x272
   TextField "Text field_1" at 11,197 size 223x43; Text 'Visiteurs max'
   TextField "Text field_2" at 14,49 size 186x43; Text 'Occupation'
   TextField "Text field_3" at 20,252 size 131x43; Text 'Alerte 1'
   TextField "Text field_4" at 20,296 size 131x43; Text 'Alerte 2'
   IOField "I/O field_2" at 234,45 size 137x53; FormatPattern 99999
      ProcessValue <- "Occupation"
   Button "Button_1" at 43,380 size 84x27; TextOff 'Modifier'; Authorization "User administration"
      on Press: function_b14e0dd5("BitModifier", 0)
      Appearance <- "AutoriseModifier"
   Button "Button_2" at 149,380 size 102x27; TextOff 'Enregistrer'
      on Press: function_b14e0dd5("BitEnregistrer", 0); function_f23ef4c9()
   Button "Button_3" at 275,380 size 84x27; TextOff 'Annuler'
      on Press: function_b14e0dd5("BitAnnuler", 0); function_f23ef4c9()
   IOField "I/O field_1" at 246,202 size 135x37; FormatPattern 99999
      ProcessValue <- "VisiteurMax"
   IOField "I/O field_3" at 245,260 size 137x32; FormatPattern 99999
      ProcessValue <- "Alerte1"
   IOField "I/O field_4" at 244,300 size 139x32; FormatPattern 99999
      ProcessValue <- "Alerte2"
   Rectangle "Rectangle_5" at 594,130 size 193x189
      Appearance <- "AnimationCarre"
   GraphicView "Graphic view_3" at 444,28 size 99x71; Picture "AlerteImage"
      Visibility <- "BitAlerte2"
   Group "Group" at 594,365 size 80x41; Picture "Up_Arrow"
   Group "Group_1" at 706,365 size 81x41; Picture "Down_Arrow"
   GraphicView "Graphic view_6" at 580,0 size 219x39; Picture "LogoFBMACASYSTEM"
   GraphicView "Graphic view_1" at 444,260 size 99x71; Picture "WarningImage"
      Visibility <- "BitAlerte1"
   GraphicView "Graphic view_2" at 426,131 size 99x71; Picture "CheckImage"
      Visibility <- "BitNoAlerte"
   Button "Button_4" at 594,365 size 80x41; TextOff 'Text'
      on Press: function_b14e0dd5("Up", 0)
      Visibility <- "AutoriseModifier"
   GraphicView "Graphic view_4" at 612,376 size 19x20; Picture "Up_Arrow"
      Visibility <- "AutoriseModifier"
   Button "Button_5" at 706,365 size 81x41; TextOff 'Text'
      on Press: function_b14e0dd5("Down", 0)
      Visibility <- "AutoriseModifier"
   GraphicView "Graphic view_5" at 725,376 size 20x20; Picture "Down_Arrow"
      Visibility <- "AutoriseModifier"
*)